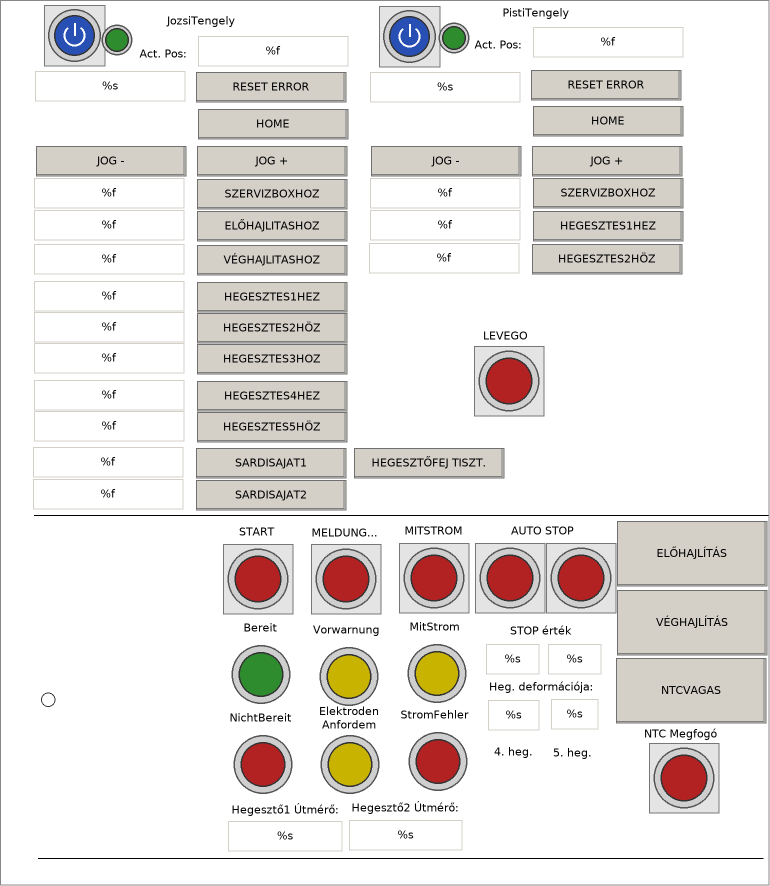
VISUALIZATION TempZoli  // 770x886
    PowerSwitch (33,5 83x61), variable: GVL.bJozsiServo, behaviour: TOGGLE, style: Switch-PowerSwitch-Blue
    Button (198,109 150x30), "HOME"
        OnMouseUp: execute { JOZSITENGELY.sJozsiAxisCommand:='HOME'; }
    Button (197,146 150x30), "JOG +"
        tap JOZSITENGELY.bJozsiJOGPlus
    Button (36,146 150x30), "JOG -"
        tap JOZSITENGELY.bJozsiJOGMinus
    Button (196,72 150x30), "RESET ERROR"
        tap JOZSITENGELY.bJozsiReset
    Textfield (35,71 150x30), "%s", text variable: JOZSITENGELY.nJozsiErrorCode, input disabled if: TRUE
    Textfield (34,210 150x30), "%f", text variable: GVL.lrHajlitoPosition1
        OnMouseClick: write the text variable via VisuDialogs.Numpad, min -10000, max -1
    Button (197,211 150x30), "ELŐHAJLITASHOZ"
        OnMouseUp: execute { JOZSITENGELY.lrJozsiPosition:=GVL.lrHajlitoPosition1; JOZSITENGELY.sJozsiAxisCommand:='MOVE'; }
    Label (88,39 150x30), "Act. Pos:"
    Textfield (198,36 150x30), "%f", text variable: JOZSITENGELY.lrJozsiActPos, input disabled if: TRUE
    Label (126,6 150x30), "JozsiTengely"
    PowerSwitch (368,6 83x61), variable: GVL.bPistiServo, behaviour: TOGGLE, style: Switch-PowerSwitch-Blue
    Button (533,106 150x30), "HOME"
        OnMouseUp: execute { PISTITENGELY.sPistiAxisCommand:='HOME'; }
    Button (532,146 150x30), "JOG +"
        tap PISTITENGELY.bPistiJOGPlus
    Button (371,146 150x30), "JOG -"
        tap PISTITENGELY.bPistiJOGMinus
    Button (531,70 150x30), "RESET ERROR"
        tap PISTITENGELY.bPistiReset
    Textfield (370,72 150x30), "%s", text variable: PISTITENGELY.nPistiErrorCode, input disabled if: TRUE
    Textfield (369,243 150x30), "%f", text variable: GVL.lrHegesztoPosition7
        OnMouseClick: write the text variable via VisuDialogs.Numpad, min -10000, max -1
    Button (532,244 150x30), "HEGESZTES2HÖZ"
        OnMouseUp: execute { PISTITENGELY.lrPistiPosition:=GVL.lrHegesztoPosition7; PISTITENGELY.sPistiAxisCommand:='MOVE'; }
    Label (423,30 150x30), "Act. Pos:"
    Textfield (533,27 150x30), "%f", text variable: PISTITENGELY.lrPistiActPos, input disabled if: TRUE
    Label (461,-2 150x30), "PistiTengely"
    Textfield (34,244 150x30), "%f", text variable: GVL.lrHajlitoPosition2
        OnMouseClick: write the text variable via VisuDialogs.Numpad, min -10000, max -1
    Button (197,245 150x30), "VÉGHAJLITASHOZ"
        OnMouseUp: execute { JOZSITENGELY.lrJozsiPosition:=GVL.lrHajlitoPosition2; JOZSITENGELY.sJozsiAxisCommand:='MOVE'; }
    Textfield (34,281 150x30), "%f", text variable: GVL.lrHegesztoPosition1
        OnMouseClick: write the text variable via VisuDialogs.Numpad, min -10000, max -1
    Button (197,282 150x30), "HEGESZTES1HEZ"
        OnMouseUp: execute { JOZSITENGELY.lrJozsiPosition:=GVL.lrHegesztoPosition1; JOZSITENGELY.sJozsiAxisCommand:='MOVE'; }
    RadioButton (39,515 150x369), variable: HEGESZTOK.nHegesztoNum
        Areas[0]: Text=Semelyik
        Areas[1]: Text=Program2HG1
        Areas[2]: Text=Program3HG1
        Areas[3]: Text=Program4HG1
        Areas[4]: Text=Program5HG2
        Areas[5]: Text=Program6HG2
        Areas[6]: Text=Program7HG3
        Areas[7]: Text=Program8HG3
    Textfield (228,821 114x30), "%s", text variable: HEGESZTOK.ulHegeszto1Utmero, input disabled if: TRUE
    Label (210,795 150x30), "Hegesztő1 Útmérő:"
    Textfield (349,820 113x30), "%s", text variable: HEGESZTOK.ulHegeszto2Utmero, input disabled if: TRUE
    Label (330,793 150x30), "Hegesztő2 Útmérő:"
    Textfield (34,312 150x30), "%f", text variable: GVL.lrHegesztoPosition2
        OnMouseClick: write the text variable via VisuDialogs.Numpad, min -10000, max -1
    Button (197,313 150x30), "HEGESZTES2HÖZ"
        OnMouseUp: execute { JOZSITENGELY.lrJozsiPosition:=GVL.lrHegesztoPosition2; JOZSITENGELY.sJozsiAxisCommand:='MOVE'; }
    Textfield (34,343 150x30), "%f", text variable: GVL.lrHegesztoPosition3
        OnMouseClick: write the text variable via VisuDialogs.Numpad, min -10000, max -1
    Button (197,344 150x30), "HEGESZTES3HOZ"
        OnMouseUp: execute { JOZSITENGELY.lrJozsiPosition:=GVL.lrHegesztoPosition3; JOZSITENGELY.sJozsiAxisCommand:='MOVE'; }
    Line (34,515) (768,515)
    PushSwitch (474,346 70x70), variable: MAIN.bLevego, behaviour: TOGGLE, style: Switch-PushSwitch-Red
    Label (471,321 69x30), "LEVEGO"
    Textfield (34,380 150x30), "%f", text variable: GVL.lrHegesztoPosition4
        OnMouseClick: write the text variable via VisuDialogs.Numpad, min -10000, max -1
    Button (197,381 150x30), "HEGESZTES4HEZ"
        OnMouseUp: execute { JOZSITENGELY.lrJozsiPosition:=GVL.lrHegesztoPosition4; JOZSITENGELY.sJozsiAxisCommand:='MOVE'; }
    Textfield (34,411 150x30), "%f", text variable: GVL.lrHegesztoPosition5
        OnMouseClick: write the text variable via VisuDialogs.Numpad, min -10000, max -1
    Button (197,412 150x30), "HEGESZTES5HÖZ"
        OnMouseUp: execute { JOZSITENGELY.lrJozsiPosition:=GVL.lrHegesztoPosition5; JOZSITENGELY.sJozsiAxisCommand:='MOVE'; }
    PushSwitch (311,544 70x70), variable: GVL.bHegesztoHibaTorles, behaviour: TOGGLE, style: Switch-PushSwitch-Red
    PushSwitch (399,543 70x70), variable: HEGESZTOK.bHegesztoMitStromOut, behaviour: TOGGLE, style: Switch-PushSwitch-Red
    PushSwitch (223,544 70x70), variable: HEGESZTOK.bHegesztoStart, behaviour: TOGGLE, style: Switch-PushSwitch-Red
    Label (222,517 69x30), "START"
    Label (310,518 69x30), "MELDUNG..."
    Label (399,516 69x30), "MITSTROM"
    Lamp1 (315,642 68x69), variable: HEGESZTOK.bHegesztoVorwarnung, style: Lamp-Lamp1-Yellow
    Label (312,615 69x30), "Vorwarnung"
    Lamp1 (316,730 68x69), variable: HEGESZTOK.bHegesztoElektrodenAnfordem, style: Lamp-Lamp1-Yellow
    Label (283,703 132x30), "Elektroden Anfordem"
    Lamp1 (227,640 68x69), variable: HEGESZTOK.bHegesztoBereit, style: Lamp-Lamp1-Green
    Label (226,613 69x30), "Bereit"
    Lamp1 (404,727 68x69), variable: HEGESZTOK.bHegesztoStromFehler, style: Lamp-Lamp1-Red
    Label (400,700 69x30), "StromFehler"
    Lamp1 (403,639 68x69), variable: HEGESZTOK.bHegesztoMitStromIn, style: Lamp-Lamp1-Yellow
    Label (400,612 69x30), "MitStrom"
    Lamp1 (229,730 68x69), variable: HEGESZTOK.bHegesztoNichtBereit, style: Lamp-Lamp1-Red
    Label (226,703 69x30), "NichtBereit"
    Line (38,858) (763,858)
    Button (617,521 150x65), "ELŐHAJLÍTÁS", input disabled if: HAJLITOK.s_InCommand <> ''
        OnMouseUp: execute {
            IF HAJLITOK.s_InCommand = '' THEN
            	HAJLITOK.s_InCommand:='ELOHAJLITAS';
            END_IF
        }
    Button (617,590 150x65), "VÉGHAJLÍTÁS", input disabled if: HAJLITOK.s_InCommand <> ''
        OnMouseUp: execute {
            IF HAJLITOK.s_InCommand = '' THEN
            	HAJLITOK.s_InCommand:='VEGHAJLITAS';
            END_IF
        }
    Button (616,658 150x65), "NTCVAGAS", input disabled if: NTCProcess.s_InCommand <> ''
        OnMouseUp: execute {
            IF NTCProcess.s_InCommand = '' THEN
            	NTCProcess.s_InCommand:='VAGAS';
            END_IF
        }
    PushSwitch (649,743 70x70), variable: NTCProcess.bMegfogo, behaviour: TOGGLE, style: Switch-PushSwitch-Red
    Label (637,719 87x30), "NTC Megfogó"
    Textfield (34,178 150x30), "%f", text variable: GVL.lrNTCSzervizbox
        OnMouseClick: write the text variable via VisuDialogs.Numpad, min -10000, max -1
    Button (197,179 150x30), "SZERVIZBOXHOZ"
        OnMouseUp: execute { JOZSITENGELY.lrJozsiPosition:=GVL.lrNTCSzervizbox; JOZSITENGELY.sJozsiAxisCommand:='MOVE'; }
    Button (533,178 150x30), "SZERVIZBOXHOZ"
        OnMouseUp: execute { PISTITENGELY.lrPistiPosition:=GVL.lrPtSzervizbox; PISTITENGELY.sPistiAxisCommand:='MOVE'; }
    Textfield (370,178 150x30), "%f", text variable: GVL.lrPtSzervizbox
        OnMouseClick: write the text variable via VisuDialogs.Numpad, min -10000, max -1
    Textfield (370,210 150x30), "%f", text variable: GVL.lrHegesztoPosition6
        OnMouseClick: write the text variable via VisuDialogs.Numpad, min -10000, max -1
    Button (533,211 150x30), "HEGESZTES1HEZ"
        OnMouseUp: execute { PISTITENGELY.lrPistiPosition:=GVL.lrHegesztoPosition6; PISTITENGELY.sPistiAxisCommand:='MOVE'; }
    Lamp1 (99,18 36x44), variable: JOZSITENGELY.bHomeReady, style: Lamp-Lamp1-Green
    Lamp1 (436,16 36x44), variable: PISTITENGELY.bHomeReady, style: Lamp-Lamp1-Green
    Textfield (33,447 150x30), "%f", text variable: JOZSITENGELY.lrSardisajatPosition1
        OnMouseClick: write the text variable via VisuDialogs.Numpad, min -10000, max -1
    Button (196,448 150x30), "SARDISAJAT1"
        OnMouseUp: execute { JOZSITENGELY.lrJozsiPosition:=JOZSITENGELY.lrSardisajatPosition1; JOZSITENGELY.sJozsiAxisCommand:='MOVE'; }
    Textfield (33,479 150x30), "%f", text variable: JOZSITENGELY.lrSardisajatPosition2
        OnMouseClick: write the text variable via VisuDialogs.Numpad, min -10000, max -1
    Button (196,480 150x30), "SARDISAJAT2"
        OnMouseUp: execute { JOZSITENGELY.lrJozsiPosition:=JOZSITENGELY.lrSardisajatPosition2; JOZSITENGELY.sJozsiAxisCommand:='MOVE'; }
    Button (354,448 150x30), "HEGESZTŐFEJ TISZT."
        OnMouseUp: execute {
            IF GVL.bJOZSITENGELYReserved=FALSE THEN
            	HEGESZTOFEJTISZTITAS.iState:=1;
            END_IF;
        }
    PushSwitch (475,543 70x70), variable: GVL.bAutomaticWeldingStop4, behaviour: TOGGLE, style: Switch-PushSwitch-Red
    Label (508,516 69x30), "AUTO STOP"
    Textfield (486,644 53x30), "%s", text variable: GVL.nWeldingStopDistance4
        OnMouseClick: write the text variable via VisuDialogs.Numpad, min 0, max 1000
    Textfield (488,700 51x30), "%s", text variable: HEGESZTESUTMERES.nWeldingDeformation4
    Label (466,672 150x30), "Heg. deformációja:"
    Textfield (551,699 47x30), "%s", text variable: HEGESZTESUTMERES.nWeldingDeformation5
    Label (502,616 78x30), "STOP érték"
    Textfield (548,644 53x30), "%s", text variable: GVL.nWeldingStopDistance5
        OnMouseClick: write the text variable via VisuDialogs.Numpad, min 0, max 1000
    PushSwitch (546,543 70x70), variable: GVL.bAutomaticWeldingStop5, behaviour: TOGGLE, style: Switch-PushSwitch-Red
    Label (491,737 45x30), "4. heg."
    Label (550,738 45x30), "5. heg."
END_VISUALIZATION

(* stored: Version 1.1.0.1, ProductVersion 3.1.4024.11
   Visu TempZoli: Id {b225fdff-f8de-4028-b9bb-4e6c340fc075} *)
